(* IEC 61131-3 sources: ATCMcontrol_Engineering/src/COM/softing/fc/AddOns/Softing/4CPCTarget/Libs/ATCM_IEC1131_3/table_22, 113 files *)

(* ---- bool_to_byte.st ---- *)
(*[[
    UserURL= "ATCM:BOOL_TO_BYTE.htm"
]]*)

FUNCTION BOOL_TO_BYTE : BYTE
VAR_INPUT
    IN : BOOL;
END_VAR

inline{%1?1:0}

END_FUNCTION

(* ---- bool_to_dint.st ---- *)
(*[[
    UserURL= "ATCM:BOOL_TO_DINT.htm"
]]*)

FUNCTION BOOL_TO_DINT : DINT
VAR_INPUT
    IN : BOOL;
END_VAR

inline{%1?1:0}

END_FUNCTION

(* ---- bool_to_dword.st ---- *)
(*[[
    UserURL= "ATCM:BOOL_TO_DWORD.htm"
]]*)

FUNCTION BOOL_TO_DWORD : DWORD
VAR_INPUT
    IN : BOOL;
END_VAR

inline{%1?1:0}

END_FUNCTION

(* ---- bool_to_int.st ---- *)
(*[[
    UserURL= "ATCM:BOOL_TO_DINT.htm"
]]*)

FUNCTION BOOL_TO_INT : INT
VAR_INPUT
    IN : BOOL;
END_VAR

inline{ VMOP(bool_to_int) }

END_FUNCTION

(* ---- bool_to_lint.st ---- *)
(*[[
    UserURL= "ATCM:BOOL_TO_LINT.htm"
]]*)

FUNCTION BOOL_TO_LINT : LINT
VAR_INPUT
    IN : BOOL;
END_VAR

inline{%1?1l:0l}

END_FUNCTION

(* ---- bool_to_lreal.st ---- *)
(*[[
    UserURL= "ATCM:BOOL_TO_LREAL.htm"
]]*)

FUNCTION BOOL_TO_LREAL : LREAL
VAR_INPUT
    IN : BOOL;
END_VAR

inline{%1?1.0:0.0}

END_FUNCTION

(* ---- bool_to_lword.st ---- *)
(*[[
    UserURL= "ATCM:BOOL_TO_LWORD.htm"
]]*)

FUNCTION BOOL_TO_LWORD : LWORD
VAR_INPUT
    IN : BOOL;
END_VAR

inline{%1?1l:0l}

END_FUNCTION

(* ---- bool_to_word.st ---- *)
(*[[
    UserURL= "ATCM:BOOL_TO_WORD.htm"
]]*)

FUNCTION BOOL_TO_WORD : WORD
VAR_INPUT
    IN : BOOL;
END_VAR

inline{%1?1:0}

END_FUNCTION

(* ---- bool_to_wstring.st ---- *)
(*[[
    UserURL= "ATCM:BOOL_TO_WSTRING.htm"
]]*)

FUNCTION BOOL_TO_WSTRING : WSTRING
VAR_INPUT
    IN : BOOL;
END_VAR

inline{%1?"TRUE":"FALSE"}

END_FUNCTION

(* ---- byte_to_bool.st ---- *)
(*[[
    UserURL= "ATCM:BYTE_TO_BOOL.htm"
]]*)

FUNCTION BYTE_TO_BOOL : BOOL
VAR_INPUT
    IN : BYTE;
END_VAR

inline{%1==0?false:true}

END_FUNCTION

(* ---- byte_to_dint.st ---- *)
(*[[
    UserURL= "ATCM:BYTE_TO_DINT.htm"
]]*)

FUNCTION BYTE_TO_DINT : DINT
VAR_INPUT
    IN : BYTE;
END_VAR

inline{%1}

END_FUNCTION

(* ---- byte_to_dword.st ---- *)
(*[[
    UserURL= "ATCM:BYTE_TO_DWORD.htm"
]]*)

FUNCTION BYTE_TO_DWORD : DWORD
VAR_INPUT
    IN : BYTE;
END_VAR

inline{%1}

END_FUNCTION

(* ---- byte_to_int.st ---- *)
(*[[
    UserURL= "ATCM:BYTE_TO_DINT.htm"
]]*)

FUNCTION BYTE_TO_INT : INT
VAR_INPUT
    IN : BYTE;
END_VAR

inline{ VMOP }

END_FUNCTION

(* ---- byte_to_lint.st ---- *)
(*[[
    UserURL= "ATCM:BYTE_TO_LINT.htm"
]]*)

FUNCTION BYTE_TO_LINT : LINT
VAR_INPUT
    IN : BYTE;
END_VAR

inline{(long)%1}

END_FUNCTION

(* ---- byte_to_lreal.st ---- *)
(*[[
    UserURL= "ATCM:BYTE_TO_LREAL.htm"
]]*)

FUNCTION BYTE_TO_LREAL : LREAL
VAR_INPUT
    IN : BYTE;
END_VAR

inline{(double)%1}

END_FUNCTION

(* ---- byte_to_lword.st ---- *)
(*[[
    UserURL= "ATCM:BYTE_TO_LWORD.htm"
]]*)

FUNCTION BYTE_TO_LWORD : LWORD
VAR_INPUT
    IN : BYTE;
END_VAR

inline{(long)%1}

END_FUNCTION

(* ---- byte_to_word.st ---- *)
(*[[
    UserURL= "ATCM:BYTE_TO_WORD.htm"
]]*)

FUNCTION BYTE_TO_WORD : WORD
VAR_INPUT
    IN : BYTE;
END_VAR

inline{%1}

END_FUNCTION

(* ---- byte_to_wstring.st ---- *)
(*[[
    UserURL= "ATCM:BYTE_TO_WSTRING.htm"
]]*)

FUNCTION BYTE_TO_WSTRING : WSTRING
VAR_INPUT
    IN : BYTE;
END_VAR

inline{java.lang.Integer.toString(%1)}

END_FUNCTION

(* ---- date_to_wstring.st ---- *)
(*[[
    UserURL= "ATCM:DATE_TO_WSTRING.htm"
]]*)

FUNCTION DATE_TO_WSTRING : WSTRING
VAR_INPUT
    IN : DATE;
END_VAR

inline{Utils.date_to_wstring(%1)}

END_FUNCTION

(* ---- dint_to_bool.st ---- *)
(*[[
    UserURL= "ATCM:DINT_TO_BOOL.htm"
]]*)

FUNCTION DINT_TO_BOOL : BOOL
VAR_INPUT
    IN : DINT;
END_VAR

inline{%1==0?false:true}

END_FUNCTION

(* ---- dint_to_byte.st ---- *)
(*[[
    UserURL= "ATCM:DINT_TO_BYTE.htm"
]]*)

FUNCTION DINT_TO_BYTE : BYTE
VAR_INPUT
    IN : DINT;
END_VAR

inline{%1&0xff}

END_FUNCTION

(* ---- dint_to_dword.st ---- *)
(*[[
    UserURL= "ATCM:DINT_TO_DWORD.htm"
]]*)

FUNCTION DINT_TO_DWORD : DWORD
VAR_INPUT
    IN : DINT;
END_VAR

inline{%1}

END_FUNCTION

(* ---- dint_to_int.st ---- *)
(*[[
    UserURL= "ATCM:DINT_TO_LINT.htm"
]]*)

FUNCTION DINT_TO_INT : INT
VAR_INPUT
    IN : DINT;
END_VAR

inline{VMOP}

END_FUNCTION

(* ---- dint_to_lint.st ---- *)
(*[[
    UserURL= "ATCM:DINT_TO_LINT.htm"
]]*)

FUNCTION DINT_TO_LINT : LINT
VAR_INPUT
    IN : DINT;
END_VAR

inline{(long)%1}

END_FUNCTION

(* ---- dint_to_lreal.st ---- *)
(*[[
    UserURL= "ATCM:DINT_TO_LREAL.htm"
]]*)

FUNCTION DINT_TO_LREAL : LREAL
VAR_INPUT
    IN : DINT;
END_VAR

inline{(double)%1}

END_FUNCTION

(* ---- dint_to_lword.st ---- *)
(*[[
    UserURL= "ATCM:DINT_TO_LWORD.htm"
]]*)

FUNCTION DINT_TO_LWORD : LWORD
VAR_INPUT
    IN : DINT;
END_VAR

inline{(long)%1}

END_FUNCTION

(* ---- dint_to_time.st ---- *)
(*[[
    UserURL= "ATCM:DINT_TO_TIME.htm"
]]*)

FUNCTION DINT_TO_TIME : TIME
VAR_INPUT
    IN : DINT;
END_VAR

inline{(long)%1}

END_FUNCTION

(* ---- dint_to_word.st ---- *)
(*[[
    UserURL= "ATCM:DINT_TO_WORD.htm"
]]*)

FUNCTION DINT_TO_WORD : WORD
VAR_INPUT
    IN : DINT;
END_VAR

inline{%1&0xffff}

END_FUNCTION

(* ---- dint_to_wstring.st ---- *)
(*[[
    UserURL= "ATCM:DINT_TO_WSTRING.htm"
]]*)

FUNCTION DINT_TO_WSTRING : WSTRING
VAR_INPUT
    IN : DINT;
END_VAR

inline{java.lang.Integer.toString(%1)}

END_FUNCTION

(* ---- dt_to_date.st ---- *)
(*[[
    UserURL= "ATCM:DT_TO_DATE.htm"
]]*)

FUNCTION DT_TO_DATE : DATE
VAR_INPUT
    IN : DT;
END_VAR

inline{Utils.dt_to_date(%1)}

END_FUNCTION

(* ---- dt_to_time.st ---- *)
(*[[
    UserURL= "ATCM:DT_TO_TIME.htm"
]]*)

FUNCTION DT_TO_TIME : TIME
VAR_INPUT
    IN : DT;
END_VAR

inline{%1}

END_FUNCTION

(* ---- dt_to_tod.st ---- *)
(*[[
    UserURL= "ATCM:DT_TO_TOD.htm"
]]*)

FUNCTION DT_TO_TOD : TOD
VAR_INPUT
    IN : DT;
END_VAR

inline{Utils.dt_to_tod(%1)}

END_FUNCTION

(* ---- dt_to_wstring.st ---- *)
(*[[
    UserURL= "ATCM:DT_TO_WSTRING.htm"
]]*)

FUNCTION DT_TO_WSTRING : WSTRING
VAR_INPUT
    IN : DT;
END_VAR

inline{Utils.dt_to_wstring(%1)}

END_FUNCTION

(* ---- dword_to_bool.st ---- *)
(*[[
    UserURL= "ATCM:DWORD_TO_BOOL.htm"
]]*)

FUNCTION DWORD_TO_BOOL : BOOL
VAR_INPUT
    IN : DWORD;
END_VAR

inline{%1==0?false:true}

END_FUNCTION

(* ---- dword_to_byte.st ---- *)
(*[[
    UserURL= "ATCM:DWORD_TO_BYTE.htm"
]]*)

FUNCTION DWORD_TO_BYTE : BYTE
VAR_INPUT
    IN : DWORD;
END_VAR

inline{%1&0xff}

END_FUNCTION

(* ---- dword_to_dint.st ---- *)
(*[[
    UserURL= "ATCM:DWORD_TO_DINT.htm"
]]*)

FUNCTION DWORD_TO_DINT : DINT
VAR_INPUT
    IN : DWORD;
END_VAR

inline{%1}

END_FUNCTION

(* ---- dword_to_int.st ---- *)
(*[[
    UserURL= "ATCM:DWORD_TO_LINT.htm"
]]*)

FUNCTION DWORD_TO_INT : INT
VAR_INPUT
    IN : DWORD;
END_VAR

inline{VMOP}

END_FUNCTION

(* ---- dword_to_lint.st ---- *)
(*[[
    UserURL= "ATCM:DWORD_TO_LINT.htm"
]]*)

FUNCTION DWORD_TO_LINT : LINT
VAR_INPUT
    IN : DWORD;
END_VAR

inline{((long)%1)&0xffffffffl}

END_FUNCTION

(* ---- dword_to_lreal.st ---- *)
(*[[
    UserURL= "ATCM:DWORD_TO_LREAL.htm"
]]*)

FUNCTION DWORD_TO_LREAL : LREAL
VAR_INPUT
    IN : DWORD;
END_VAR

inline{(double)(0x00000000ffffffffL & %1)}

END_FUNCTION

(* ---- dword_to_lword.st ---- *)
(*[[
    UserURL= "ATCM:DWORD_TO_LWORD.htm"
]]*)

FUNCTION DWORD_TO_LWORD : LWORD
VAR_INPUT
    IN : DWORD;
END_VAR

inline{((long)%1)&0xffffffffl}

END_FUNCTION

(* ---- dword_to_word.st ---- *)
(*[[
    UserURL= "ATCM:DWORD_TO_WORD.htm"
]]*)

FUNCTION DWORD_TO_WORD : WORD
VAR_INPUT
    IN : DWORD;
END_VAR

inline{%1&0xffff}

END_FUNCTION

(* ---- dword_to_wstring.st ---- *)
(*[[
    UserURL= "ATCM:DWORD_TO_WSTRING.htm"
]]*)

FUNCTION DWORD_TO_WSTRING : WSTRING
VAR_INPUT
    IN : DWORD;
END_VAR

inline{java.lang.Long.toString(0x00000000ffffffffL & %1)}

END_FUNCTION

(* ---- int_to_bool.st ---- *)
(*[[
    UserURL= "ATCM:DINT_TO_BOOL.htm"
]]*)

FUNCTION INT_TO_BOOL : BOOL
VAR_INPUT
    IN : INT;
END_VAR

inline{VMOP(WORD_TO_BOOL)}

END_FUNCTION

(* ---- int_to_byte.st ---- *)
(*[[
    UserURL= "ATCM:DINT_TO_BYTE.htm"
]]*)

FUNCTION INT_TO_BYTE : BYTE
VAR_INPUT
    IN : INT;
END_VAR

inline{VMOP(word_to_byte
; int_to_byte
; push word#16#ff
; and_word
)
      }

END_FUNCTION

(* ---- int_to_dint.st ---- *)
(*[[
    UserURL= "ATCM:DINT_TO_LINT.htm"
]]*)

FUNCTION INT_TO_DINT : DINT
VAR_INPUT
    IN : INT;
END_VAR

inline{VMOP}

END_FUNCTION

(* ---- int_to_dword.st ---- *)
(*[[
    UserURL= "ATCM:DINT_TO_DWORD.htm"
]]*)

FUNCTION INT_TO_DWORD : DWORD
VAR_INPUT
    IN : INT;
END_VAR

inline{VMOP}

END_FUNCTION

(* ---- int_to_lint.st ---- *)
(*[[
    UserURL= "ATCM:DINT_TO_LINT.htm"
]]*)

FUNCTION INT_TO_LINT : LINT
VAR_INPUT
    IN : INT;
END_VAR

inline{VMOP}

END_FUNCTION

(* ---- int_to_lreal.st ---- *)
(*[[
    UserURL= "ATCM:DINT_TO_LREAL.htm"
]]*)

FUNCTION INT_TO_LREAL : LREAL
VAR_INPUT
    IN : INT;
END_VAR

inline{VMOP}

END_FUNCTION

(* ---- int_to_real.st ---- *)
(*[[
    UserURL= "ATCM:DINT_TO_LREAL.htm"
]]*)

FUNCTION INT_TO_REAL : REAL
VAR_INPUT
    IN : INT;
END_VAR

inline{VMOP}

END_FUNCTION

(* ---- int_to_string.st ---- *)
(*[[
    UserURL= "ATCM:DINT_TO_WSTRING.htm"
]]*)

FUNCTION INT_TO_STRING : STRING
VAR_INPUT
    IN : INT;
END_VAR

inline{ STDLIB(int_to_string) }

END_FUNCTION

(* ---- int_to_time.st ---- *)
(*[[
    UserURL= "ATCM:DINT_TO_TIME.htm"
]]*)

FUNCTION INT_TO_TIME : TIME
VAR_INPUT
    IN : INT;
END_VAR

inline
{
	%1
	int_to_dint
}

END_FUNCTION

(* ---- int_to_word.st ---- *)
(*[[
    UserURL= "ATCM:DINT_TO_WORD.htm"
]]*)

FUNCTION INT_TO_WORD : WORD
VAR_INPUT
    IN : INT;
END_VAR

inline{NOOP}

END_FUNCTION

(* ---- lint_to_bool.st ---- *)
(*[[
    UserURL= "ATCM:LINT_TO_BOOL.htm"
]]*)

FUNCTION LINT_TO_BOOL : BOOL
VAR_INPUT
    IN : LINT;
END_VAR

inline{%1==0l?false:true}

END_FUNCTION

(* ---- lint_to_byte.st ---- *)
(*[[
    UserURL= "ATCM:LINT_TO_BYTE.htm"
]]*)

FUNCTION LINT_TO_BYTE : BYTE
VAR_INPUT
    IN : LINT;
END_VAR

inline{(int)%1&0xff}

END_FUNCTION

(* ---- lint_to_dint.st ---- *)
(*[[
    UserURL= "ATCM:LINT_TO_DINT.htm"
]]*)

FUNCTION LINT_TO_DINT : DINT
VAR_INPUT
    IN : LINT;
END_VAR

inline{(int)%1}

END_FUNCTION

(* ---- lint_to_dword.st ---- *)
(*[[
    UserURL= "ATCM:LINT_TO_DWORD.htm"
]]*)

FUNCTION LINT_TO_DWORD : DWORD
VAR_INPUT
    IN : LINT;
END_VAR

inline{(int)%1}

END_FUNCTION

(* ---- lint_to_int.st ---- *)
(*[[
    UserURL= "ATCM:LINT_TO_DINT.htm"
]]*)

FUNCTION LINT_TO_INT : INT
VAR_INPUT
    IN : LINT;
END_VAR

inline{(int)%1}

END_FUNCTION

(* ---- lint_to_lreal.st ---- *)
(*[[
    UserURL= "ATCM:LINT_TO_LREAL.htm"
]]*)

FUNCTION LINT_TO_LREAL : LREAL
VAR_INPUT
    IN : LINT;
END_VAR

inline{(double)%1}

END_FUNCTION

(* ---- lint_to_lword.st ---- *)
(*[[
    UserURL= "ATCM:LINT_TO_LWORD.htm"
]]*)

FUNCTION LINT_TO_LWORD : LWORD
VAR_INPUT
    IN : LINT;
END_VAR

inline{%1}

END_FUNCTION

(* ---- lint_to_time.st ---- *)
(*[[
    UserURL= "ATCM:LINT_TO_TIME.htm"
]]*)

FUNCTION LINT_TO_TIME : TIME
VAR_INPUT
    IN : LINT;
END_VAR

inline{%1}

END_FUNCTION

(* ---- lint_to_word.st ---- *)
(*[[
    UserURL= "ATCM:LINT_TO_WORD.htm"
]]*)

FUNCTION LINT_TO_WORD : WORD
VAR_INPUT
    IN : LINT;
END_VAR

inline{(int)%1&0xffff}

END_FUNCTION

(* ---- lint_to_wstring.st ---- *)
(*[[
    UserURL= "ATCM:LINT_TO_WSTRING.htm"
]]*)

FUNCTION LINT_TO_WSTRING : WSTRING
VAR_INPUT
    IN : LINT;
END_VAR

inline{java.lang.Long.toString(%1)}

END_FUNCTION

(* ---- lreal_to_bool.st ---- *)
(*[[
    UserURL= "ATCM:LREAL_TO_BOOL.htm"
]]*)

FUNCTION LREAL_TO_BOOL : BOOL
VAR_INPUT
    IN : LREAL;
END_VAR

inline{%1==0.0?false:true}

END_FUNCTION

(* ---- lreal_to_byte.st ---- *)
(*[[
    UserURL= "ATCM:LREAL_TO_BYTE.htm"
]]*)

FUNCTION LREAL_TO_BYTE : BYTE
VAR_INPUT
    IN : LREAL;
END_VAR

inline{((int)Math.round(%1))&0xff}

END_FUNCTION

(* ---- lreal_to_dint.st ---- *)
(*[[
    UserURL= "ATCM:LREAL_TO_DINT.htm"
]]*)

FUNCTION LREAL_TO_DINT : DINT
VAR_INPUT
    IN : LREAL;
END_VAR

inline{Utils.doubleToIntIEC599(%1)}

END_FUNCTION

(* ---- lreal_to_dword.st ---- *)
(*[[
    UserURL= "ATCM:LREAL_TO_DWORD.htm"
]]*)

FUNCTION LREAL_TO_DWORD : DWORD
VAR_INPUT
    IN : LREAL;
END_VAR

inline{(int)Math.round(%1)}

END_FUNCTION

(* ---- lreal_to_int.st ---- *)
(*[[
    UserURL= "ATCM:LREAL_TO_LINT.htm"
]]*)

FUNCTION LREAL_TO_INT : INT
VAR_INPUT
    IN : LREAL;
END_VAR

inline{VMOP}

END_FUNCTION

(* ---- lreal_to_lint.st ---- *)
(*[[
    UserURL= "ATCM:LREAL_TO_LINT.htm"
]]*)

FUNCTION LREAL_TO_LINT : LINT
VAR_INPUT
    IN : LREAL;
END_VAR

inline{Utils.doubleToLongIEC599(%1)}

END_FUNCTION

(* ---- lreal_to_lword.st ---- *)
(*
 * Note:
 *  LREAL_TO_LWORD(x) is the same as
 *  LINT_TO_LWORD(LREAL_TO_LINT(x))
 *
 *  e.g.  LREAL_TO_LWORD(-1.0E0) = 16#ffffffffffffffff;
 *)

FUNCTION LREAL_TO_LWORD : LWORD
VAR_INPUT
    IN : LREAL;
END_VAR

inline{Math.round(%1)}

END_FUNCTION

(* ---- lreal_to_time.st ---- *)
(*[[
    UserURL= "ATCM:LREAL_TO_TIME.htm"
]]*)

FUNCTION LREAL_TO_TIME : TIME
VAR_INPUT
    IN : LREAL;
END_VAR

inline{(long)%1}

END_FUNCTION

(* ---- lreal_to_word.st ---- *)
(*[[
    UserURL= "ATCM:LREAL_TO_WORD.htm"
]]*)

FUNCTION LREAL_TO_WORD : WORD
VAR_INPUT
    IN : LREAL;
END_VAR

inline{((int)Math.round(%1))&0xffff}

END_FUNCTION

(* ---- lreal_to_wstring.st ---- *)
(*[[
    UserURL= "ATCM:LREAL_TO_WSTRING.htm"
]]*)

FUNCTION LREAL_TO_WSTRING : WSTRING
VAR_INPUT
    IN : LREAL;
END_VAR

inline{java.lang.Double.toString(%1)}

END_FUNCTION

(* ---- lword_to_bool.st ---- *)
(*[[
    UserURL= "ATCM:LWORD_TO_BOOL.htm"
]]*)

FUNCTION LWORD_TO_BOOL : BOOL
VAR_INPUT
    IN : LWORD;
END_VAR

inline{%1==0l?false:true}

END_FUNCTION

(* ---- lword_to_byte.st ---- *)
(*[[
    UserURL= "ATCM:LWORD_TO_BYTE.htm"
]]*)

FUNCTION LWORD_TO_BYTE : BYTE
VAR_INPUT
    IN : LWORD;
END_VAR

inline{(int)%1&0xff}

END_FUNCTION

(* ---- lword_to_dint.st ---- *)
(*[[
    UserURL= "ATCM:LWORD_TO_DINT.htm"
]]*)

FUNCTION LWORD_TO_DINT : DINT
VAR_INPUT
    IN : LWORD;
END_VAR

inline{(int)%1}

END_FUNCTION

(* ---- lword_to_dword.st ---- *)
(*[[
    UserURL= "ATCM:LWORD_TO_DWORD.htm"
]]*)

FUNCTION LWORD_TO_DWORD : DWORD
VAR_INPUT
    IN : LWORD;
END_VAR

inline{(int)%1}

END_FUNCTION

(* ---- lword_to_int.st ---- *)
(*[[
    UserURL= "ATCM:LWORD_TO_DINT.htm"
]]*)

FUNCTION LWORD_TO_INT : INT
VAR_INPUT
    IN : LWORD;
END_VAR

inline{(int)%1}

END_FUNCTION

(* ---- lword_to_lint.st ---- *)
(*[[
    UserURL= "ATCM:LWORD_TO_LINT.htm"
]]*)

FUNCTION LWORD_TO_LINT : LINT
VAR_INPUT
    IN : LWORD;
END_VAR

inline{%1}

END_FUNCTION

(* ---- lword_to_lreal.st ---- *)
(*
 * Note:
 *  LWORD_TO_LREAL(x) is the same as
 *  LINT_TO_LREAL(LWORD_TO_LINT(x))
 *
 *  e.g.  LWORD_TO_LREAL(16#ffffffffffffffff) = -1.0E0
 *)
FUNCTION LWORD_TO_LREAL : LREAL
VAR_INPUT
    IN : LWORD;
END_VAR

inline{(double)%1}

END_FUNCTION

(* ---- lword_to_word.st ---- *)
(*[[
    UserURL= "ATCM:LWORD_TO_WORD.htm"
]]*)

FUNCTION LWORD_TO_WORD : WORD
VAR_INPUT
    IN : LWORD;
END_VAR

inline{(int)%1&0xffff}

END_FUNCTION

(* ---- lword_to_wstring.st ---- *)
(*[[
    UserURL= "ATCM:LWORD_TO_WSTRING.htm"
]]*)

FUNCTION LWORD_TO_WSTRING : WSTRING
VAR_INPUT
    IN : LWORD;
END_VAR

inline{Utils.lword_to_wstring(%1)}

END_FUNCTION

(* ---- real_to_int.st ---- *)
(*[[
    UserURL= "ATCM:REAL_TO_INT.htm"
]]*)

FUNCTION REAL_TO_INT : INT
VAR_INPUT
    IN : REAL;
END_VAR

inline{VMOP}

END_FUNCTION

(* ---- string_to_int.st ---- *)
(*[[
    UserURL= "ATCM:WSTRING_TO_LINT.htm"
]]*)

FUNCTION STRING_TO_INT : INT
VAR_INPUT
    IN : STRING;
END_VAR

inline{ STDLIB(string_to_int) }

END_FUNCTION

(* ---- time_to_dint.st ---- *)
(*[[
    UserURL= "ATCM:TIME_TO_DINT.htm",
    deprecated="to avoid unexpected truncation use TIME_TO_LINT instead"
]]*)

FUNCTION TIME_TO_DINT : DINT
VAR_INPUT
    IN : TIME;
END_VAR

inline{(int)%1}

END_FUNCTION

(* ---- time_to_dt.st ---- *)
(*[[
    UserURL= "ATCM:TIME_TO_DT.htm"
]]*)

FUNCTION TIME_TO_DT : DT
VAR_INPUT
    IN : TIME;
END_VAR

inline{%1}

END_FUNCTION

(* ---- time_to_int.st ---- *)
(*[[
    UserURL= "ATCM:TIME_TO_LINT.htm"
]]*)

FUNCTION TIME_TO_INT : INT
VAR_INPUT
    IN : TIME;
END_VAR

inline
{
    %1
    dint_to_int
}

END_FUNCTION

(* ---- time_to_lint.st ---- *)
(*[[
    UserURL= "ATCM:TIME_TO_LINT.htm"
]]*)

FUNCTION TIME_TO_LINT : LINT
VAR_INPUT
    IN : TIME;
END_VAR

inline{%1}

END_FUNCTION

(* ---- time_to_lreal.st ---- *)
(*[[
    UserURL= "ATCM:TIME_TO_LREAL.htm"
]]*)

FUNCTION TIME_TO_LREAL : LREAL
VAR_INPUT
    IN : TIME;
END_VAR

inline{(double)%1}

END_FUNCTION

(* ---- time_to_wstring.st ---- *)
(*[[
    UserURL= "ATCM:TIME_TO_WSTRING.htm"
]]*)

FUNCTION TIME_TO_WSTRING : WSTRING
VAR_INPUT
   IN : TIME;
END_VAR

inline{"t#"+java.lang.Long.toString(%1)+"ms"}

END_FUNCTION

(* ---- tod_to_time.st ---- *)
(*[[
    UserURL= "ATCM:TOD_TO_TIME.htm"
]]*)

FUNCTION TOD_TO_TIME : TIME
VAR_INPUT
    IN : TOD;
END_VAR

inline{(long)%1}

END_FUNCTION

(* ---- tod_to_wstring.st ---- *)
(*[[
    UserURL= "ATCM:TOD_TO_WSTRING.htm"
]]*)

FUNCTION TOD_TO_WSTRING : WSTRING
VAR_INPUT
    IN : TOD;
END_VAR

inline{Utils.tod_to_wstring(%1)}

END_FUNCTION

(* ---- trunc.st ---- *)
(*[[
    UserURL= "ATCM:TRUNC.htm"
]]*)

FUNCTION TRUNC : ANY_INT
VAR_INPUT
    IN : ANY_REAL;
END_VAR

overload DINT(ANY_REAL) inline{(int)%1}
overload LINT(ANY_REAL) inline{(long)%1}

END_FUNCTION

(* ---- word_to_bool.st ---- *)
(*[[
    UserURL= "ATCM:WORD_TO_BOOL.htm"
]]*)

FUNCTION WORD_TO_BOOL : BOOL
VAR_INPUT
    IN : WORD;
END_VAR

inline{%1==0?false:true}

END_FUNCTION

(* ---- word_to_byte.st ---- *)
(*[[
    UserURL= "ATCM:WORD_TO_BYTE.htm"
]]*)

FUNCTION WORD_TO_BYTE : BYTE
VAR_INPUT
    IN : WORD;
END_VAR

inline{%1&0xff}

END_FUNCTION

(* ---- word_to_dint.st ---- *)
(*[[
    UserURL= "ATCM:WORD_TO_DINT.htm"
]]*)

FUNCTION WORD_TO_DINT : DINT
VAR_INPUT
    IN : WORD;
END_VAR

inline{%1}

END_FUNCTION

(* ---- word_to_dword.st ---- *)
(*[[
    UserURL= "ATCM:WORD_TO_DWORD.htm"
]]*)

FUNCTION WORD_TO_DWORD : DWORD
VAR_INPUT
    IN : WORD;
END_VAR

inline{%1}

END_FUNCTION

(* ---- word_to_int.st ---- *)
(*[[
    UserURL= "ATCM:WORD_TO_INT.htm"
]]*)

FUNCTION WORD_TO_INT : INT
VAR_INPUT
    IN : WORD;
END_VAR

inline{NOOP}

END_FUNCTION

(* ---- word_to_lint.st ---- *)
(*[[
    UserURL= "ATCM:WORD_TO_LINT.htm"
]]*)

FUNCTION WORD_TO_LINT : LINT
VAR_INPUT
    IN : WORD;
END_VAR

inline{(long)%1}

END_FUNCTION

(* ---- word_to_lreal.st ---- *)
(*[[
    UserURL= "ATCM:WORD_TO_LREAL.htm"
]]*)

FUNCTION WORD_TO_LREAL : LREAL
VAR_INPUT
    IN : WORD;
END_VAR

inline{(double)%1}

END_FUNCTION

(* ---- word_to_lword.st ---- *)
(*[[
    UserURL= "ATCM:WORD_TO_LWORD.htm"
]]*)

FUNCTION WORD_TO_LWORD : LWORD
VAR_INPUT
    IN : WORD;
END_VAR

inline{(long)%1}

END_FUNCTION

(* ---- word_to_wstring.st ---- *)
(*[[
    UserURL= "ATCM:WORD_TO_WSTRING.htm"
]]*)

FUNCTION WORD_TO_WSTRING : WSTRING
VAR_INPUT
    IN : WORD;
END_VAR

inline{java.lang.Integer.toString(%1)}

END_FUNCTION

(* ---- wstring_to_bool.st ---- *)
(*[[
    UserURL= "ATCM:WSTRING_TO_BOOL.htm"
]]*)

FUNCTION WSTRING_TO_BOOL : BOOL
VAR_INPUT
    IN : WSTRING;
END_VAR

inline{Utils.wstring_to_bool(tc,%1)}

END_FUNCTION

(* ---- wstring_to_byte.st ---- *)
(*[[
    UserURL= "ATCM:WSTRING_TO_BYTE.htm"
]]*)

FUNCTION WSTRING_TO_BYTE : BYTE
VAR_INPUT
    IN : WSTRING;
END_VAR

inline{Utils.wstring_to_byte(tc,%1)}

END_FUNCTION

(* ---- wstring_to_date.st ---- *)
(*[[
    UserURL= "ATCM:WSTRING_TO_DATE.htm"
]]*)

FUNCTION WSTRING_TO_DATE : DATE
VAR_INPUT
    IN : WSTRING;
END_VAR

inline{Utils.wstring_to_date(tc,%1)}

END_FUNCTION

(* ---- wstring_to_dint.st ---- *)
(*[[
    UserURL= "ATCM:WSTRING_TO_DINT.htm"
]]*)

FUNCTION WSTRING_TO_DINT : DINT
VAR_INPUT
    IN : WSTRING;
END_VAR

inline{Utils.wstring_to_dint(tc,%1)}

END_FUNCTION

(* ---- wstring_to_dt.st ---- *)
(*[[
    UserURL= "ATCM:WSTRING_TO_DT.htm"
]]*)

FUNCTION WSTRING_TO_DT : DT
VAR_INPUT
    IN : WSTRING;
END_VAR

inline{Utils.wstring_to_dt(tc,%1)}

END_FUNCTION

(* ---- wstring_to_dword.st ---- *)
(*[[
    UserURL= "ATCM:WSTRING_TO_DWORD.htm"
]]*)

FUNCTION WSTRING_TO_DWORD : DWORD
VAR_INPUT
    IN : WSTRING;
END_VAR

inline{Utils.wstring_to_dword(tc,%1)}

END_FUNCTION

(* ---- wstring_to_lint.st ---- *)
(*[[
    UserURL= "ATCM:WSTRING_TO_LINT.htm"
]]*)

FUNCTION WSTRING_TO_LINT : LINT
VAR_INPUT
    IN : WSTRING;
END_VAR

inline{Utils.wstring_to_lint(tc,%1)}

END_FUNCTION

(* ---- wstring_to_lreal.st ---- *)
(*[[
    UserURL= "ATCM:WSTRING_TO_LREAL.htm"
]]*)

FUNCTION WSTRING_TO_LREAL : LREAL
VAR_INPUT
    IN : WSTRING;
END_VAR

inline{Utils.wstring_to_lreal(tc,%1)}

END_FUNCTION

(* ---- wstring_to_lword.st ---- *)
(*[[
    UserURL= "ATCM:WSTRING_TO_LWORD.htm"
]]*)

FUNCTION WSTRING_TO_LWORD : LWORD
VAR_INPUT
    IN : WSTRING;
END_VAR

inline{Utils.wstring_to_lword(tc,%1)}

END_FUNCTION

(* ---- wstring_to_time.st ---- *)
(*[[
    UserURL= "ATCM:WSTRING_TO_TIME.htm"
]]*)

FUNCTION WSTRING_TO_TIME : TIME
VAR_INPUT
    IN : WSTRING;
END_VAR

inline{Utils.wstring_to_time(tc,%1)}

END_FUNCTION

(* ---- wstring_to_tod.st ---- *)
(*[[
    UserURL= "ATCM:WSTRING_TO_TOD.htm"
]]*)

FUNCTION WSTRING_TO_TOD : TOD
VAR_INPUT
    IN : WSTRING;
END_VAR

inline{Utils.wstring_to_tod(tc,%1)}

END_FUNCTION

(* ---- wstring_to_word.st ---- *)
(*[[
    UserURL= "ATCM:WSTRING_TO_WORD.htm"
]]*)

FUNCTION WSTRING_TO_WORD : WORD
VAR_INPUT
    IN : WSTRING;
END_VAR

inline{Utils.wstring_to_word(tc,%1)}

END_FUNCTION
